Fanuc KAREL source: kt00372.KL

PROGRAM KT00372
%STACKSIZE=65535
%PRIORITY=65535
%NOLOCKGROUP
VAR
R1 : REAL
OUT : BOOLEAN
-- UNRESOLVED DECLARATIONS (source type spelling not recovered)
-- H2 : ARRAY[2] OF TYPE_0x0017 (type_u16=0x2017)
BEGIN
R1=2.0
-- UNRESOLVED_PC line 9 opcodes [2E 22 9D 33 B4] marker_code=16
-- UNRESOLVED_PC line 10 opcodes [21 22 9D 33 B3 64 70 23] marker_code=35
END KT00372
